// Mitsubishi GX Works2 project: ST_FB_NEW   PLC: Q02U

PROGRAM DIO
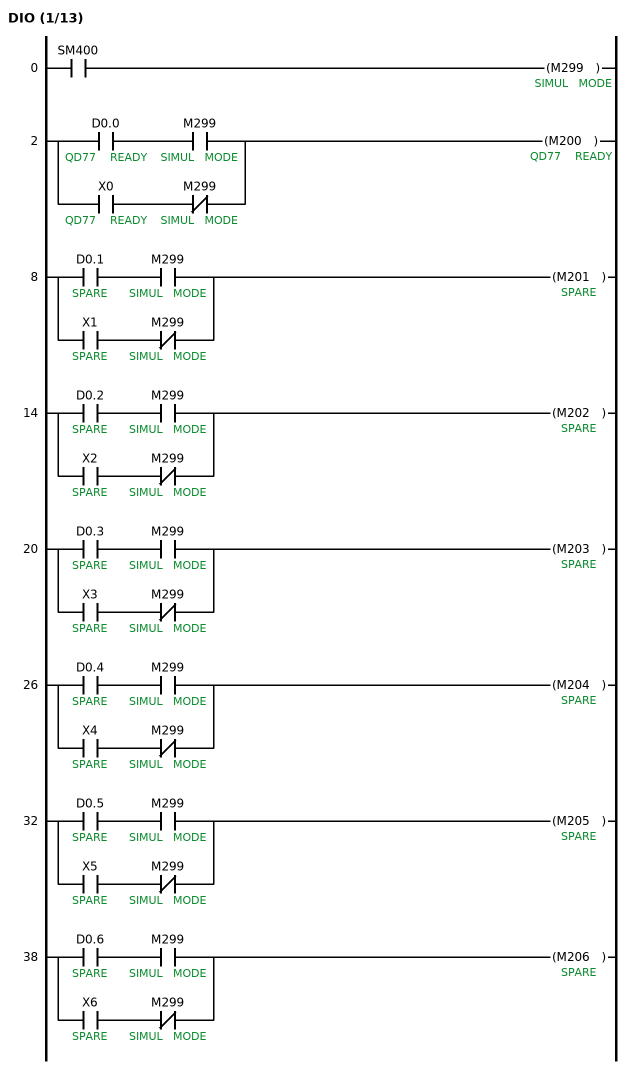
0     LD      SM400
      OUT     M299  ; SIMUL   MODE
2     LD      D0.0  ; QD77    READY
      AND     M299  ; SIMUL   MODE
      LD      X0  ; QD77    READY
      ANI     M299  ; SIMUL   MODE
      ORB
      OUT     M200  ; QD77    READY
8     LD      D0.1  ; SPARE
      AND     M299  ; SIMUL   MODE
      LD      X1  ; SPARE
      ANI     M299  ; SIMUL   MODE
      ORB
      OUT     M201  ; SPARE
14    LD      D0.2  ; SPARE
      AND     M299  ; SIMUL   MODE
      LD      X2  ; SPARE
      ANI     M299  ; SIMUL   MODE
      ORB
      OUT     M202  ; SPARE
20    LD      D0.3  ; SPARE
      AND     M299  ; SIMUL   MODE
      LD      X3  ; SPARE
      ANI     M299  ; SIMUL   MODE
      ORB
      OUT     M203  ; SPARE
26    LD      D0.4  ; SPARE
      AND     M299  ; SIMUL   MODE
      LD      X4  ; SPARE
      ANI     M299  ; SIMUL   MODE
      ORB
      OUT     M204  ; SPARE
32    LD      D0.5  ; SPARE
      AND     M299  ; SIMUL   MODE
      LD      X5  ; SPARE
      ANI     M299  ; SIMUL   MODE
      ORB
      OUT     M205  ; SPARE
38    LD      D0.6  ; SPARE
      AND     M299  ; SIMUL   MODE
      LD      X6  ; SPARE
      ANI     M299  ; SIMUL   MODE
      ORB
      OUT     M206  ; SPARE
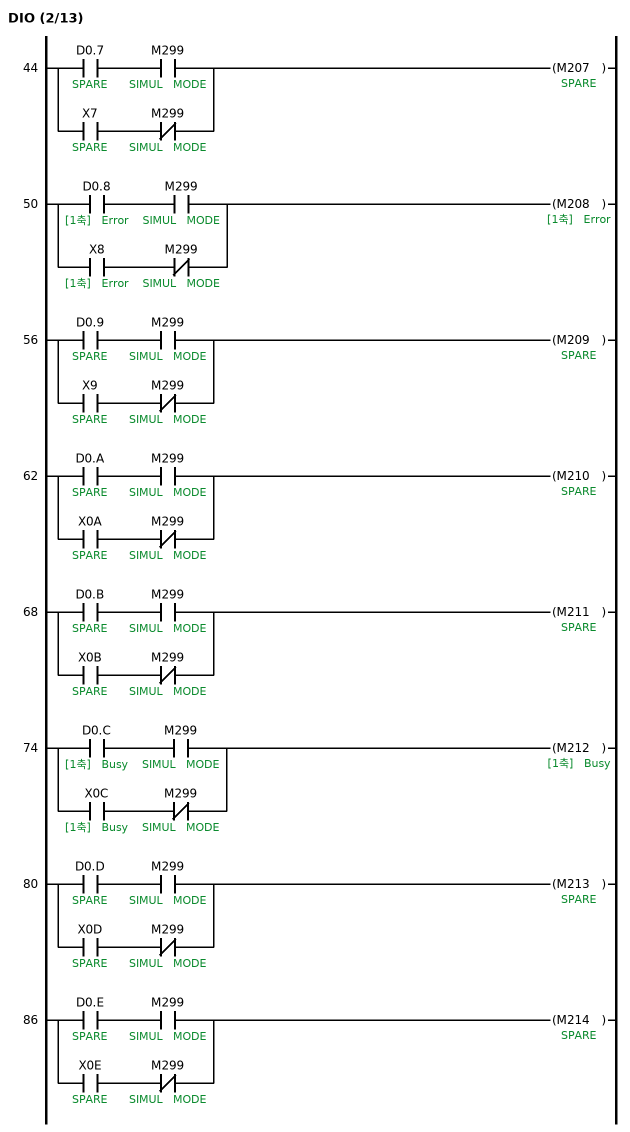
44    LD      D0.7  ; SPARE
      AND     M299  ; SIMUL   MODE
      LD      X7  ; SPARE
      ANI     M299  ; SIMUL   MODE
      ORB
      OUT     M207  ; SPARE
50    LD      D0.8  ; [1축]   Error
      AND     M299  ; SIMUL   MODE
      LD      X8  ; [1축]   Error
      ANI     M299  ; SIMUL   MODE
      ORB
      OUT     M208  ; [1축]   Error
56    LD      D0.9  ; SPARE
      AND     M299  ; SIMUL   MODE
      LD      X9  ; SPARE
      ANI     M299  ; SIMUL   MODE
      ORB
      OUT     M209  ; SPARE
62    LD      D0.A  ; SPARE
      AND     M299  ; SIMUL   MODE
      LD      X0A  ; SPARE
      ANI     M299  ; SIMUL   MODE
      ORB
      OUT     M210  ; SPARE
68    LD      D0.B  ; SPARE
      AND     M299  ; SIMUL   MODE
      LD      X0B  ; SPARE
      ANI     M299  ; SIMUL   MODE
      ORB
      OUT     M211  ; SPARE
74    LD      D0.C  ; [1축]   Busy
      AND     M299  ; SIMUL   MODE
      LD      X0C  ; [1축]   Busy
      ANI     M299  ; SIMUL   MODE
      ORB
      OUT     M212  ; [1축]   Busy
80    LD      D0.D  ; SPARE
      AND     M299  ; SIMUL   MODE
      LD      X0D  ; SPARE
      ANI     M299  ; SIMUL   MODE
      ORB
      OUT     M213  ; SPARE
86    LD      D0.E  ; SPARE
      AND     M299  ; SIMUL   MODE
      LD      X0E  ; SPARE
      ANI     M299  ; SIMUL   MODE
      ORB
      OUT     M214  ; SPARE
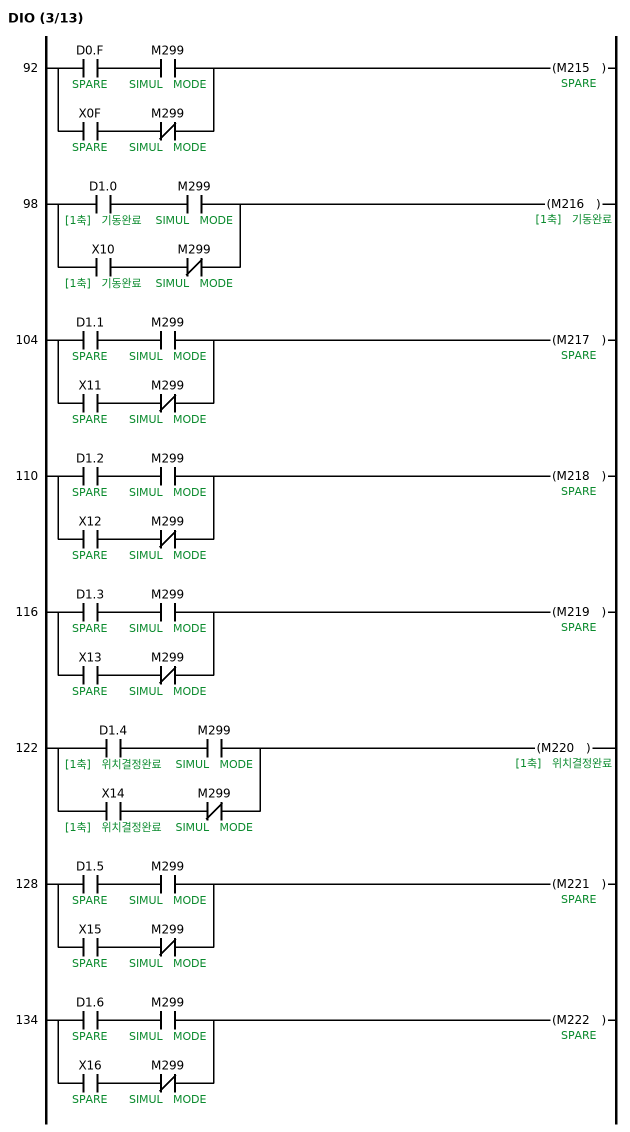
92    LD      D0.F  ; SPARE
      AND     M299  ; SIMUL   MODE
      LD      X0F  ; SPARE
      ANI     M299  ; SIMUL   MODE
      ORB
      OUT     M215  ; SPARE
98    LD      D1.0  ; [1축]   기동완료
      AND     M299  ; SIMUL   MODE
      LD      X10  ; [1축]   기동완료
      ANI     M299  ; SIMUL   MODE
      ORB
      OUT     M216  ; [1축]   기동완료
104   LD      D1.1  ; SPARE
      AND     M299  ; SIMUL   MODE
      LD      X11  ; SPARE
      ANI     M299  ; SIMUL   MODE
      ORB
      OUT     M217  ; SPARE
110   LD      D1.2  ; SPARE
      AND     M299  ; SIMUL   MODE
      LD      X12  ; SPARE
      ANI     M299  ; SIMUL   MODE
      ORB
      OUT     M218  ; SPARE
116   LD      D1.3  ; SPARE
      AND     M299  ; SIMUL   MODE
      LD      X13  ; SPARE
      ANI     M299  ; SIMUL   MODE
      ORB
      OUT     M219  ; SPARE
122   LD      D1.4  ; [1축]   위치결정완료
      AND     M299  ; SIMUL   MODE
      LD      X14  ; [1축]   위치결정완료
      ANI     M299  ; SIMUL   MODE
      ORB
      OUT     M220  ; [1축]   위치결정완료
128   LD      D1.5  ; SPARE
      AND     M299  ; SIMUL   MODE
      LD      X15  ; SPARE
      ANI     M299  ; SIMUL   MODE
      ORB
      OUT     M221  ; SPARE
134   LD      D1.6  ; SPARE
      AND     M299  ; SIMUL   MODE
      LD      X16  ; SPARE
      ANI     M299  ; SIMUL   MODE
      ORB
      OUT     M222  ; SPARE
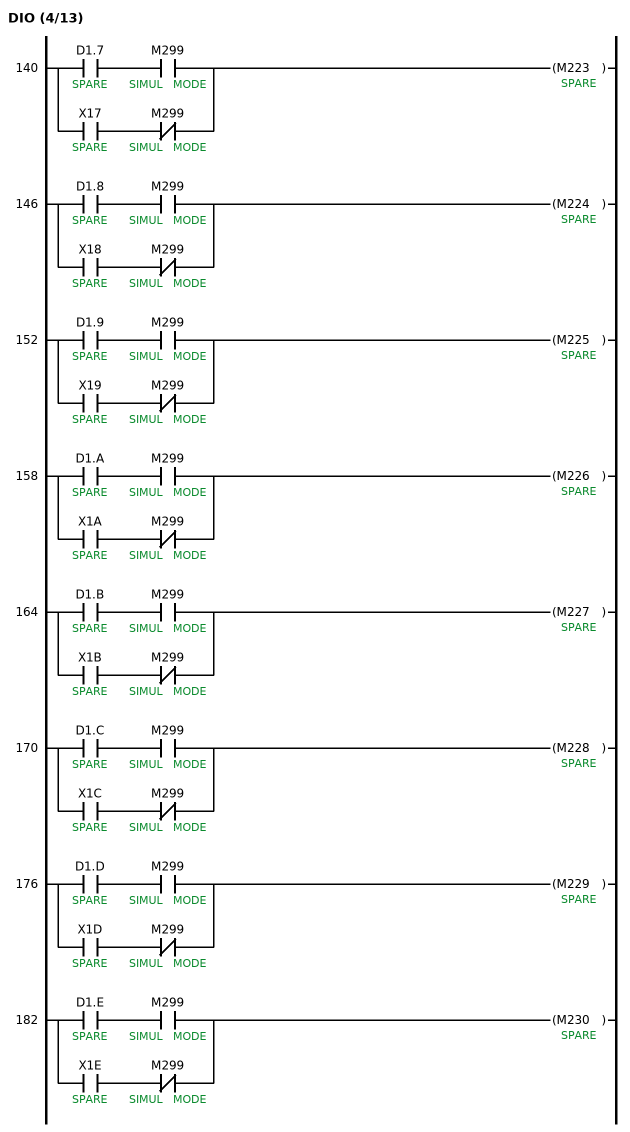
140   LD      D1.7  ; SPARE
      AND     M299  ; SIMUL   MODE
      LD      X17  ; SPARE
      ANI     M299  ; SIMUL   MODE
      ORB
      OUT     M223  ; SPARE
146   LD      D1.8  ; SPARE
      AND     M299  ; SIMUL   MODE
      LD      X18  ; SPARE
      ANI     M299  ; SIMUL   MODE
      ORB
      OUT     M224  ; SPARE
152   LD      D1.9  ; SPARE
      AND     M299  ; SIMUL   MODE
      LD      X19  ; SPARE
      ANI     M299  ; SIMUL   MODE
      ORB
      OUT     M225  ; SPARE
158   LD      D1.A  ; SPARE
      AND     M299  ; SIMUL   MODE
      LD      X1A  ; SPARE
      ANI     M299  ; SIMUL   MODE
      ORB
      OUT     M226  ; SPARE
164   LD      D1.B  ; SPARE
      AND     M299  ; SIMUL   MODE
      LD      X1B  ; SPARE
      ANI     M299  ; SIMUL   MODE
      ORB
      OUT     M227  ; SPARE
170   LD      D1.C  ; SPARE
      AND     M299  ; SIMUL   MODE
      LD      X1C  ; SPARE
      ANI     M299  ; SIMUL   MODE
      ORB
      OUT     M228  ; SPARE
176   LD      D1.D  ; SPARE
      AND     M299  ; SIMUL   MODE
      LD      X1D  ; SPARE
      ANI     M299  ; SIMUL   MODE
      ORB
      OUT     M229  ; SPARE
182   LD      D1.E  ; SPARE
      AND     M299  ; SIMUL   MODE
      LD      X1E  ; SPARE
      ANI     M299  ; SIMUL   MODE
      ORB
      OUT     M230  ; SPARE
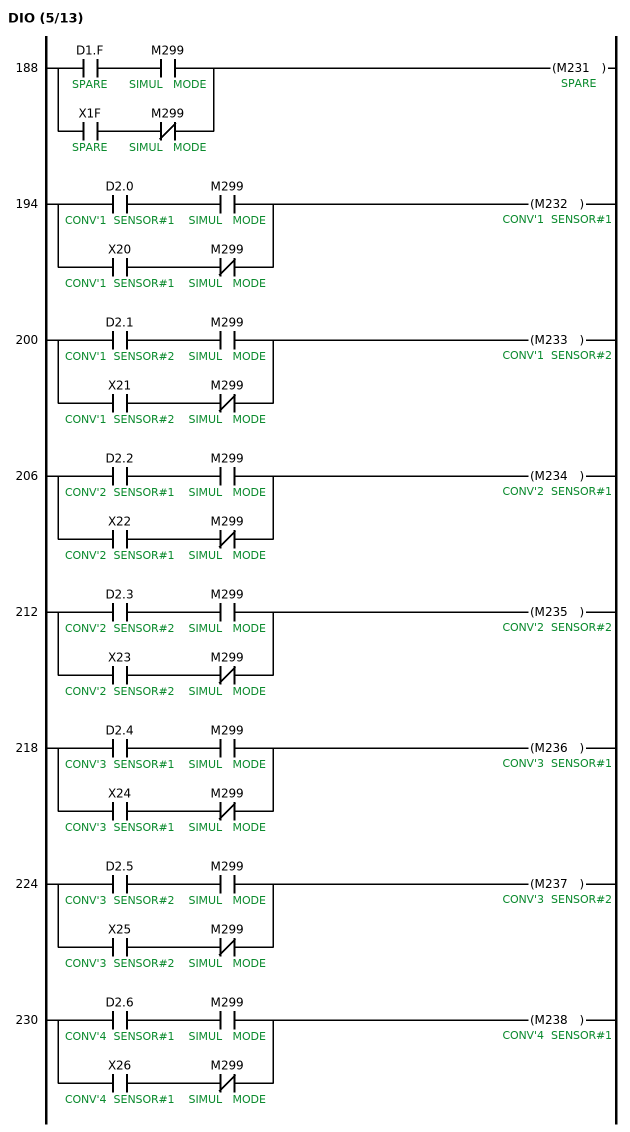
188   LD      D1.F  ; SPARE
      AND     M299  ; SIMUL   MODE
      LD      X1F  ; SPARE
      ANI     M299  ; SIMUL   MODE
      ORB
      OUT     M231  ; SPARE
194   LD      D2.0  ; CONV'1  SENSOR#1
      AND     M299  ; SIMUL   MODE
      LD      X20  ; CONV'1  SENSOR#1
      ANI     M299  ; SIMUL   MODE
      ORB
      OUT     M232  ; CONV'1  SENSOR#1
200   LD      D2.1  ; CONV'1  SENSOR#2
      AND     M299  ; SIMUL   MODE
      LD      X21  ; CONV'1  SENSOR#2
      ANI     M299  ; SIMUL   MODE
      ORB
      OUT     M233  ; CONV'1  SENSOR#2
206   LD      D2.2  ; CONV'2  SENSOR#1
      AND     M299  ; SIMUL   MODE
      LD      X22  ; CONV'2  SENSOR#1
      ANI     M299  ; SIMUL   MODE
      ORB
      OUT     M234  ; CONV'2  SENSOR#1
212   LD      D2.3  ; CONV'2  SENSOR#2
      AND     M299  ; SIMUL   MODE
      LD      X23  ; CONV'2  SENSOR#2
      ANI     M299  ; SIMUL   MODE
      ORB
      OUT     M235  ; CONV'2  SENSOR#2
218   LD      D2.4  ; CONV'3  SENSOR#1
      AND     M299  ; SIMUL   MODE
      LD      X24  ; CONV'3  SENSOR#1
      ANI     M299  ; SIMUL   MODE
      ORB
      OUT     M236  ; CONV'3  SENSOR#1
224   LD      D2.5  ; CONV'3  SENSOR#2
      AND     M299  ; SIMUL   MODE
      LD      X25  ; CONV'3  SENSOR#2
      ANI     M299  ; SIMUL   MODE
      ORB
      OUT     M237  ; CONV'3  SENSOR#2
230   LD      D2.6  ; CONV'4  SENSOR#1
      AND     M299  ; SIMUL   MODE
      LD      X26  ; CONV'4  SENSOR#1
      ANI     M299  ; SIMUL   MODE
      ORB
      OUT     M238  ; CONV'4  SENSOR#1
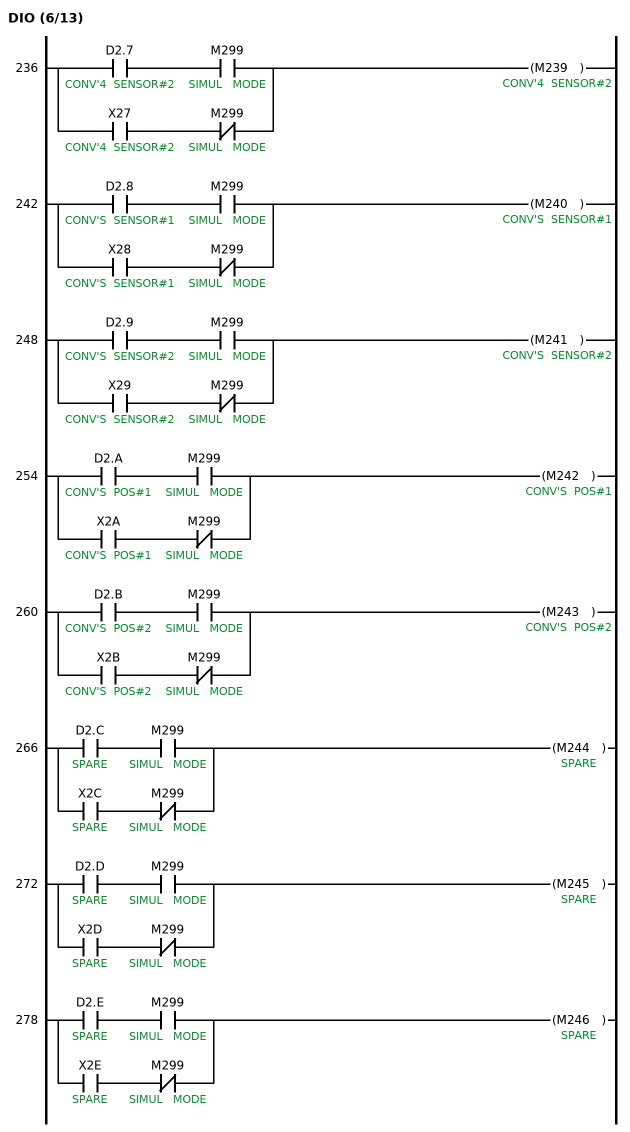
236   LD      D2.7  ; CONV'4  SENSOR#2
      AND     M299  ; SIMUL   MODE
      LD      X27  ; CONV'4  SENSOR#2
      ANI     M299  ; SIMUL   MODE
      ORB
      OUT     M239  ; CONV'4  SENSOR#2
242   LD      D2.8  ; CONV'S  SENSOR#1
      AND     M299  ; SIMUL   MODE
      LD      X28  ; CONV'S  SENSOR#1
      ANI     M299  ; SIMUL   MODE
      ORB
      OUT     M240  ; CONV'S  SENSOR#1
248   LD      D2.9  ; CONV'S  SENSOR#2
      AND     M299  ; SIMUL   MODE
      LD      X29  ; CONV'S  SENSOR#2
      ANI     M299  ; SIMUL   MODE
      ORB
      OUT     M241  ; CONV'S  SENSOR#2
254   LD      D2.A  ; CONV'S  POS#1
      AND     M299  ; SIMUL   MODE
      LD      X2A  ; CONV'S  POS#1
      ANI     M299  ; SIMUL   MODE
      ORB
      OUT     M242  ; CONV'S  POS#1
260   LD      D2.B  ; CONV'S  POS#2
      AND     M299  ; SIMUL   MODE
      LD      X2B  ; CONV'S  POS#2
      ANI     M299  ; SIMUL   MODE
      ORB
      OUT     M243  ; CONV'S  POS#2
266   LD      D2.C  ; SPARE
      AND     M299  ; SIMUL   MODE
      LD      X2C  ; SPARE
      ANI     M299  ; SIMUL   MODE
      ORB
      OUT     M244  ; SPARE
272   LD      D2.D  ; SPARE
      AND     M299  ; SIMUL   MODE
      LD      X2D  ; SPARE
      ANI     M299  ; SIMUL   MODE
      ORB
      OUT     M245  ; SPARE
278   LD      D2.E  ; SPARE
      AND     M299  ; SIMUL   MODE
      LD      X2E  ; SPARE
      ANI     M299  ; SIMUL   MODE
      ORB
      OUT     M246  ; SPARE
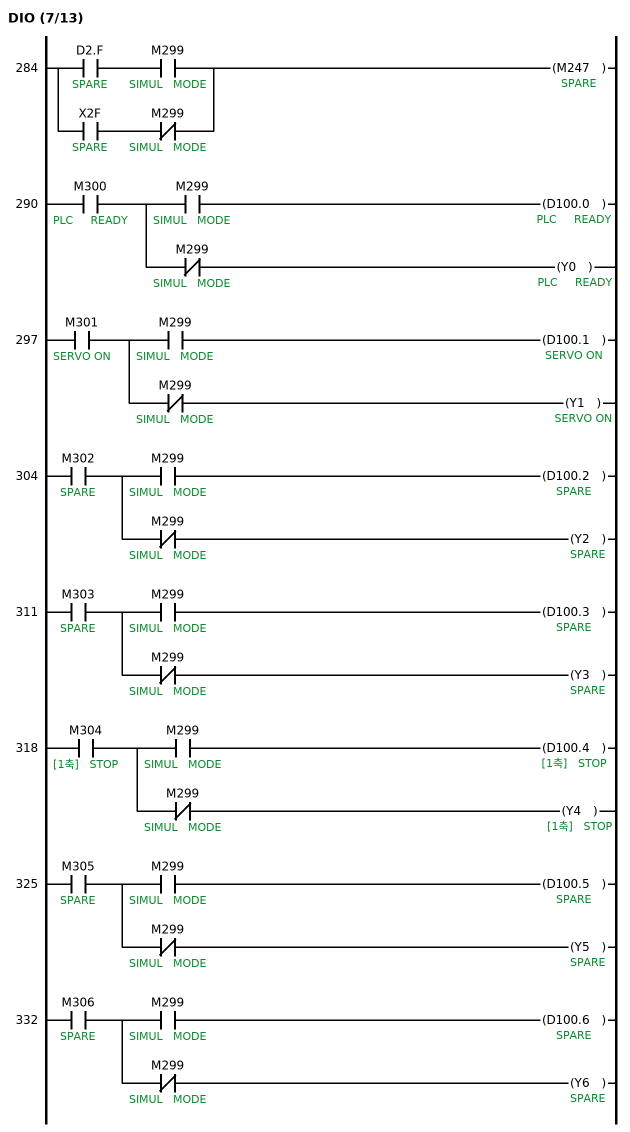
284   LD      D2.F  ; SPARE
      AND     M299  ; SIMUL   MODE
      LD      X2F  ; SPARE
      ANI     M299  ; SIMUL   MODE
      ORB
      OUT     M247  ; SPARE
290   LD      M300  ; PLC     READY
      MPS
      AND     M299  ; SIMUL   MODE
      OUT     D100.0  ; PLC     READY
      MPP
      ANI     M299  ; SIMUL   MODE
      OUT     Y0  ; PLC     READY
297   LD      M301  ; SERVO ON
      MPS
      AND     M299  ; SIMUL   MODE
      OUT     D100.1  ; SERVO ON
      MPP
      ANI     M299  ; SIMUL   MODE
      OUT     Y1  ; SERVO ON
304   LD      M302  ; SPARE
      MPS
      AND     M299  ; SIMUL   MODE
      OUT     D100.2  ; SPARE
      MPP
      ANI     M299  ; SIMUL   MODE
      OUT     Y2  ; SPARE
311   LD      M303  ; SPARE
      MPS
      AND     M299  ; SIMUL   MODE
      OUT     D100.3  ; SPARE
      MPP
      ANI     M299  ; SIMUL   MODE
      OUT     Y3  ; SPARE
318   LD      M304  ; [1축]   STOP
      MPS
      AND     M299  ; SIMUL   MODE
      OUT     D100.4  ; [1축]   STOP
      MPP
      ANI     M299  ; SIMUL   MODE
      OUT     Y4  ; [1축]   STOP
325   LD      M305  ; SPARE
      MPS
      AND     M299  ; SIMUL   MODE
      OUT     D100.5  ; SPARE
      MPP
      ANI     M299  ; SIMUL   MODE
      OUT     Y5  ; SPARE
332   LD      M306  ; SPARE
      MPS
      AND     M299  ; SIMUL   MODE
      OUT     D100.6  ; SPARE
      MPP
      ANI     M299  ; SIMUL   MODE
      OUT     Y6  ; SPARE
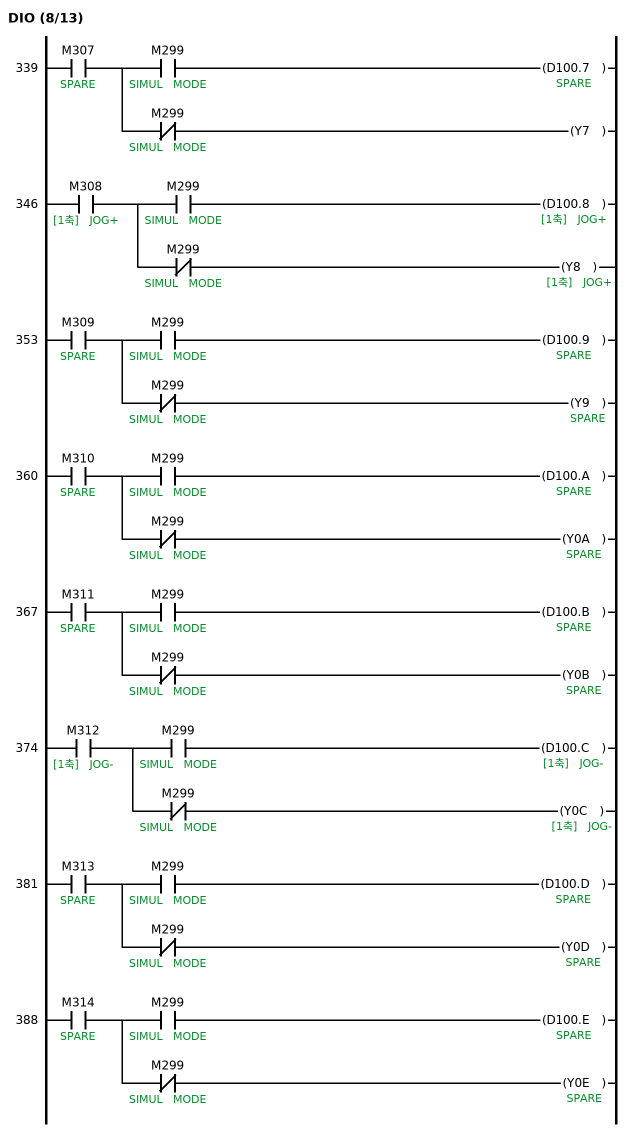
339   LD      M307  ; SPARE
      MPS
      AND     M299  ; SIMUL   MODE
      OUT     D100.7  ; SPARE
      MPP
      ANI     M299  ; SIMUL   MODE
      OUT     Y7
346   LD      M308  ; [1축]   JOG+
      MPS
      AND     M299  ; SIMUL   MODE
      OUT     D100.8  ; [1축]   JOG+
      MPP
      ANI     M299  ; SIMUL   MODE
      OUT     Y8  ; [1축]   JOG+
353   LD      M309  ; SPARE
      MPS
      AND     M299  ; SIMUL   MODE
      OUT     D100.9  ; SPARE
      MPP
      ANI     M299  ; SIMUL   MODE
      OUT     Y9  ; SPARE
360   LD      M310  ; SPARE
      MPS
      AND     M299  ; SIMUL   MODE
      OUT     D100.A  ; SPARE
      MPP
      ANI     M299  ; SIMUL   MODE
      OUT     Y0A  ; SPARE
367   LD      M311  ; SPARE
      MPS
      AND     M299  ; SIMUL   MODE
      OUT     D100.B  ; SPARE
      MPP
      ANI     M299  ; SIMUL   MODE
      OUT     Y0B  ; SPARE
374   LD      M312  ; [1축]   JOG-
      MPS
      AND     M299  ; SIMUL   MODE
      OUT     D100.C  ; [1축]   JOG-
      MPP
      ANI     M299  ; SIMUL   MODE
      OUT     Y0C  ; [1축]   JOG-
381   LD      M313  ; SPARE
      MPS
      AND     M299  ; SIMUL   MODE
      OUT     D100.D  ; SPARE
      MPP
      ANI     M299  ; SIMUL   MODE
      OUT     Y0D  ; SPARE
388   LD      M314  ; SPARE
      MPS
      AND     M299  ; SIMUL   MODE
      OUT     D100.E  ; SPARE
      MPP
      ANI     M299  ; SIMUL   MODE
      OUT     Y0E  ; SPARE
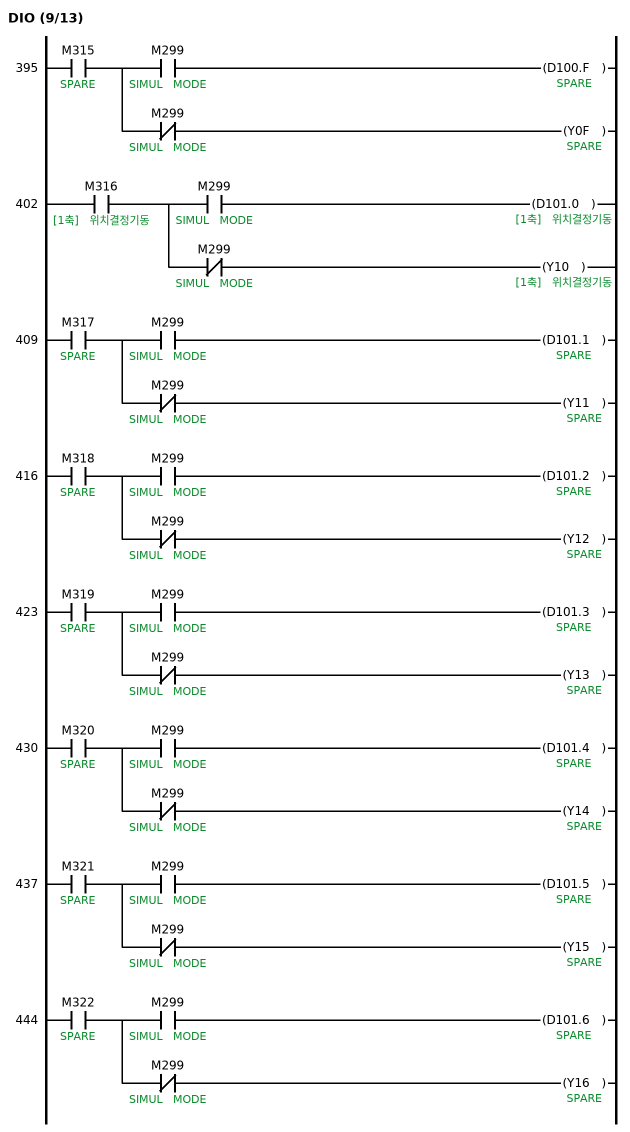
395   LD      M315  ; SPARE
      MPS
      AND     M299  ; SIMUL   MODE
      OUT     D100.F  ; SPARE
      MPP
      ANI     M299  ; SIMUL   MODE
      OUT     Y0F  ; SPARE
402   LD      M316  ; [1축]   위치결정기동
      MPS
      AND     M299  ; SIMUL   MODE
      OUT     D101.0  ; [1축]   위치결정기동
      MPP
      ANI     M299  ; SIMUL   MODE
      OUT     Y10  ; [1축]   위치결정기동
409   LD      M317  ; SPARE
      MPS
      AND     M299  ; SIMUL   MODE
      OUT     D101.1  ; SPARE
      MPP
      ANI     M299  ; SIMUL   MODE
      OUT     Y11  ; SPARE
416   LD      M318  ; SPARE
      MPS
      AND     M299  ; SIMUL   MODE
      OUT     D101.2  ; SPARE
      MPP
      ANI     M299  ; SIMUL   MODE
      OUT     Y12  ; SPARE
423   LD      M319  ; SPARE
      MPS
      AND     M299  ; SIMUL   MODE
      OUT     D101.3  ; SPARE
      MPP
      ANI     M299  ; SIMUL   MODE
      OUT     Y13  ; SPARE
430   LD      M320  ; SPARE
      MPS
      AND     M299  ; SIMUL   MODE
      OUT     D101.4  ; SPARE
      MPP
      ANI     M299  ; SIMUL   MODE
      OUT     Y14  ; SPARE
437   LD      M321  ; SPARE
      MPS
      AND     M299  ; SIMUL   MODE
      OUT     D101.5  ; SPARE
      MPP
      ANI     M299  ; SIMUL   MODE
      OUT     Y15  ; SPARE
444   LD      M322  ; SPARE
      MPS
      AND     M299  ; SIMUL   MODE
      OUT     D101.6  ; SPARE
      MPP
      ANI     M299  ; SIMUL   MODE
      OUT     Y16  ; SPARE
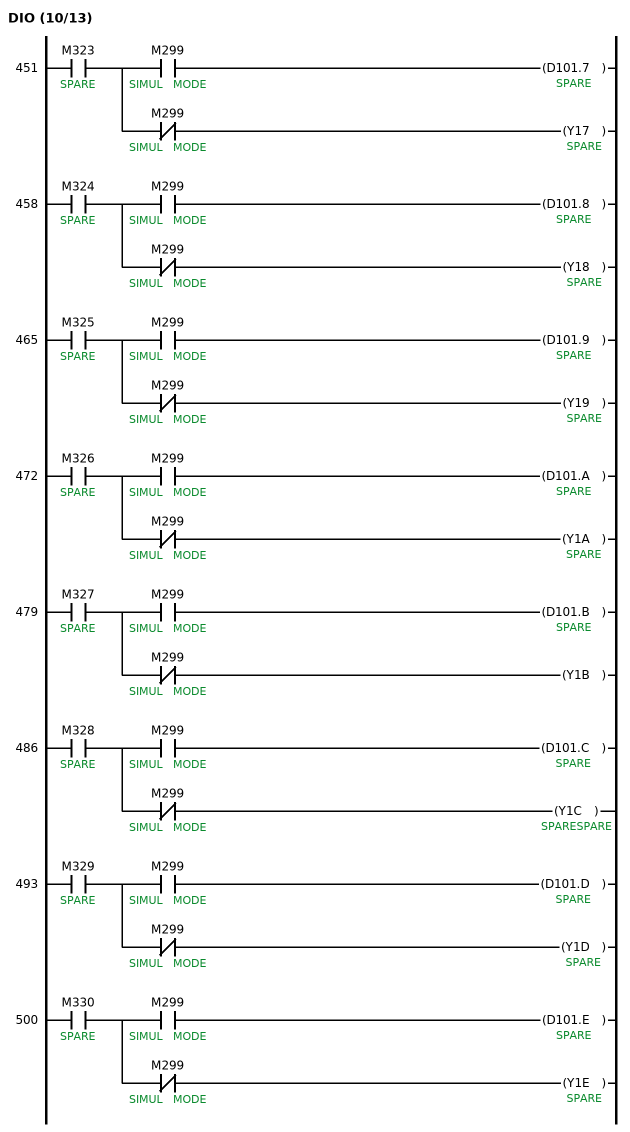
451   LD      M323  ; SPARE
      MPS
      AND     M299  ; SIMUL   MODE
      OUT     D101.7  ; SPARE
      MPP
      ANI     M299  ; SIMUL   MODE
      OUT     Y17  ; SPARE
458   LD      M324  ; SPARE
      MPS
      AND     M299  ; SIMUL   MODE
      OUT     D101.8  ; SPARE
      MPP
      ANI     M299  ; SIMUL   MODE
      OUT     Y18  ; SPARE
465   LD      M325  ; SPARE
      MPS
      AND     M299  ; SIMUL   MODE
      OUT     D101.9  ; SPARE
      MPP
      ANI     M299  ; SIMUL   MODE
      OUT     Y19  ; SPARE
472   LD      M326  ; SPARE
      MPS
      AND     M299  ; SIMUL   MODE
      OUT     D101.A  ; SPARE
      MPP
      ANI     M299  ; SIMUL   MODE
      OUT     Y1A  ; SPARE
479   LD      M327  ; SPARE
      MPS
      AND     M299  ; SIMUL   MODE
      OUT     D101.B  ; SPARE
      MPP
      ANI     M299  ; SIMUL   MODE
      OUT     Y1B
486   LD      M328  ; SPARE
      MPS
      AND     M299  ; SIMUL   MODE
      OUT     D101.C  ; SPARE
      MPP
      ANI     M299  ; SIMUL   MODE
      OUT     Y1C  ; SPARESPARE
493   LD      M329  ; SPARE
      MPS
      AND     M299  ; SIMUL   MODE
      OUT     D101.D  ; SPARE
      MPP
      ANI     M299  ; SIMUL   MODE
      OUT     Y1D  ; SPARE
500   LD      M330  ; SPARE
      MPS
      AND     M299  ; SIMUL   MODE
      OUT     D101.E  ; SPARE
      MPP
      ANI     M299  ; SIMUL   MODE
      OUT     Y1E  ; SPARE
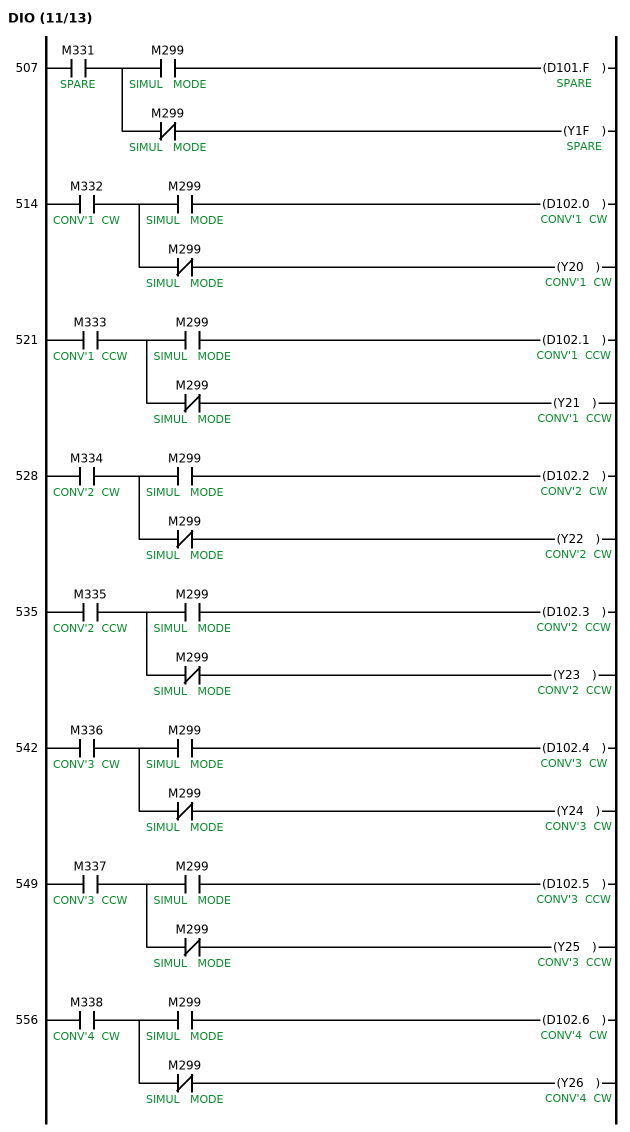
507   LD      M331  ; SPARE
      MPS
      AND     M299  ; SIMUL   MODE
      OUT     D101.F  ; SPARE
      MPP
      ANI     M299  ; SIMUL   MODE
      OUT     Y1F  ; SPARE
514   LD      M332  ; CONV'1  CW
      MPS
      AND     M299  ; SIMUL   MODE
      OUT     D102.0  ; CONV'1  CW
      MPP
      ANI     M299  ; SIMUL   MODE
      OUT     Y20  ; CONV'1  CW
521   LD      M333  ; CONV'1  CCW
      MPS
      AND     M299  ; SIMUL   MODE
      OUT     D102.1  ; CONV'1  CCW
      MPP
      ANI     M299  ; SIMUL   MODE
      OUT     Y21  ; CONV'1  CCW
528   LD      M334  ; CONV'2  CW
      MPS
      AND     M299  ; SIMUL   MODE
      OUT     D102.2  ; CONV'2  CW
      MPP
      ANI     M299  ; SIMUL   MODE
      OUT     Y22  ; CONV'2  CW
535   LD      M335  ; CONV'2  CCW
      MPS
      AND     M299  ; SIMUL   MODE
      OUT     D102.3  ; CONV'2  CCW
      MPP
      ANI     M299  ; SIMUL   MODE
      OUT     Y23  ; CONV'2  CCW
542   LD      M336  ; CONV'3  CW
      MPS
      AND     M299  ; SIMUL   MODE
      OUT     D102.4  ; CONV'3  CW
      MPP
      ANI     M299  ; SIMUL   MODE
      OUT     Y24  ; CONV'3  CW
549   LD      M337  ; CONV'3  CCW
      MPS
      AND     M299  ; SIMUL   MODE
      OUT     D102.5  ; CONV'3  CCW
      MPP
      ANI     M299  ; SIMUL   MODE
      OUT     Y25  ; CONV'3  CCW
556   LD      M338  ; CONV'4  CW
      MPS
      AND     M299  ; SIMUL   MODE
      OUT     D102.6  ; CONV'4  CW
      MPP
      ANI     M299  ; SIMUL   MODE
      OUT     Y26  ; CONV'4  CW
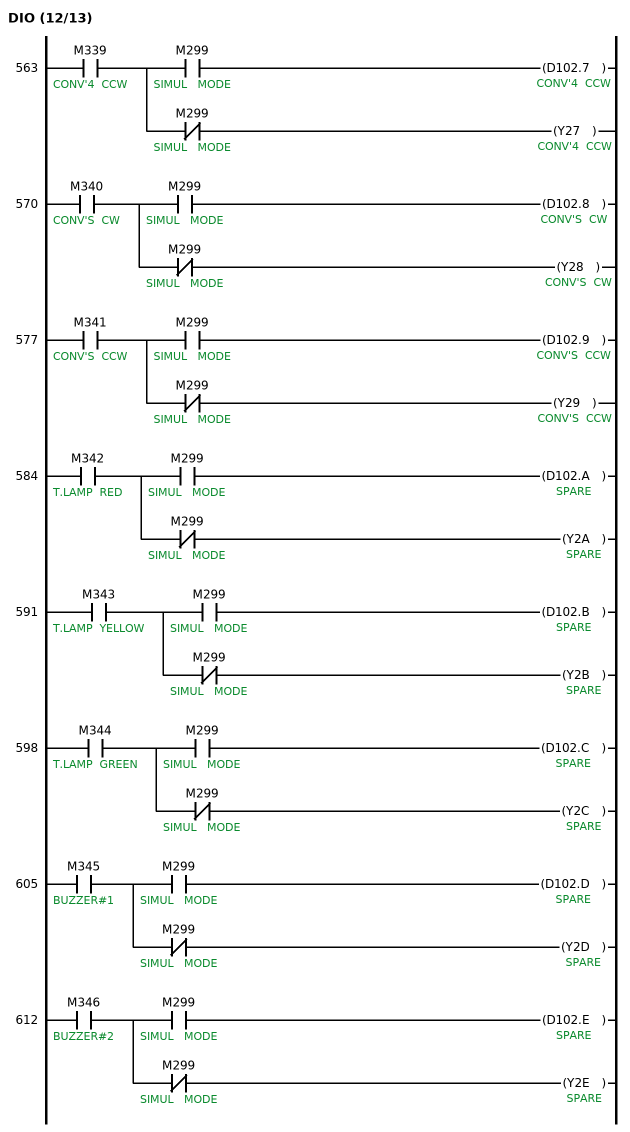
563   LD      M339  ; CONV'4  CCW
      MPS
      AND     M299  ; SIMUL   MODE
      OUT     D102.7  ; CONV'4  CCW
      MPP
      ANI     M299  ; SIMUL   MODE
      OUT     Y27  ; CONV'4  CCW
570   LD      M340  ; CONV'S  CW
      MPS
      AND     M299  ; SIMUL   MODE
      OUT     D102.8  ; CONV'S  CW
      MPP
      ANI     M299  ; SIMUL   MODE
      OUT     Y28  ; CONV'S  CW
577   LD      M341  ; CONV'S  CCW
      MPS
      AND     M299  ; SIMUL   MODE
      OUT     D102.9  ; CONV'S  CCW
      MPP
      ANI     M299  ; SIMUL   MODE
      OUT     Y29  ; CONV'S  CCW
584   LD      M342  ; T.LAMP  RED
      MPS
      AND     M299  ; SIMUL   MODE
      OUT     D102.A  ; SPARE
      MPP
      ANI     M299  ; SIMUL   MODE
      OUT     Y2A  ; SPARE
591   LD      M343  ; T.LAMP  YELLOW
      MPS
      AND     M299  ; SIMUL   MODE
      OUT     D102.B  ; SPARE
      MPP
      ANI     M299  ; SIMUL   MODE
      OUT     Y2B  ; SPARE
598   LD      M344  ; T.LAMP  GREEN
      MPS
      AND     M299  ; SIMUL   MODE
      OUT     D102.C  ; SPARE
      MPP
      ANI     M299  ; SIMUL   MODE
      OUT     Y2C  ; SPARE
605   LD      M345  ; BUZZER#1
      MPS
      AND     M299  ; SIMUL   MODE
      OUT     D102.D  ; SPARE
      MPP
      ANI     M299  ; SIMUL   MODE
      OUT     Y2D  ; SPARE
612   LD      M346  ; BUZZER#2
      MPS
      AND     M299  ; SIMUL   MODE
      OUT     D102.E  ; SPARE
      MPP
      ANI     M299  ; SIMUL   MODE
      OUT     Y2E  ; SPARE
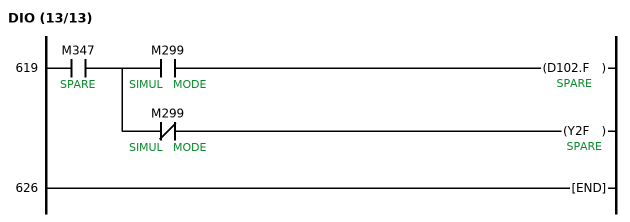
619   LD      M347  ; SPARE
      MPS
      AND     M299  ; SIMUL   MODE
      OUT     D102.F  ; SPARE
      MPP
      ANI     M299  ; SIMUL   MODE
      OUT     Y2F  ; SPARE
626   END
END_PROGRAM

PROGRAM SERVO
VAR
  SERVO_FB_1 : SERVO_FB;
END_VAR
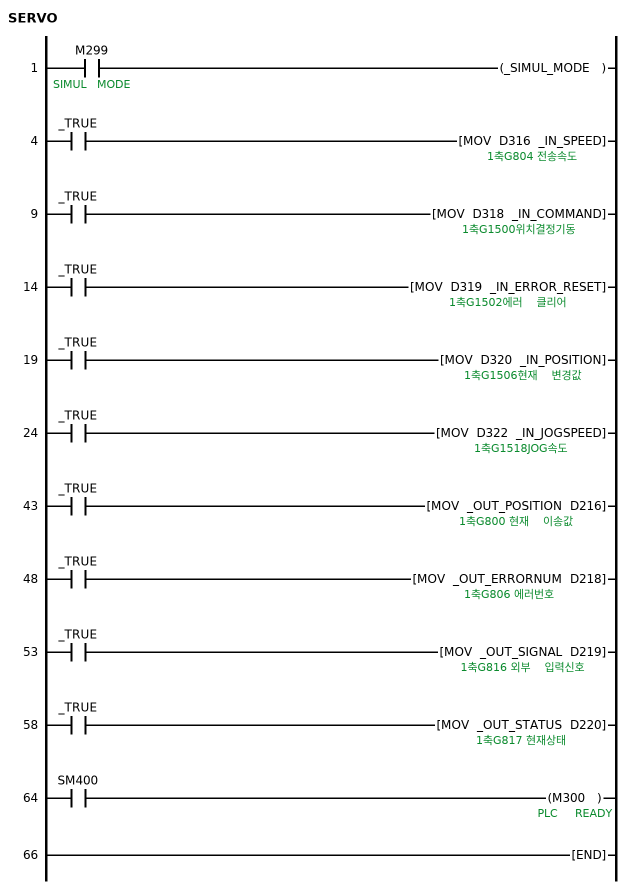
; FB BLK START SERVO_FB(SERVO_FB_1)
1     LD      M299  ; SIMUL   MODE
      OUT     _SIMUL_MODE
4     LD      _TRUE
      MOV     D316 _IN_SPEED  ; 1축G804 전송속도
9     LD      _TRUE
      MOV     D318 _IN_COMMAND  ; 1축G1500위치결정기동
14    LD      _TRUE
      MOV     D319 _IN_ERROR_RESET  ; 1축G1502에러    클리어
19    LD      _TRUE
      MOV     D320 _IN_POSITION  ; 1축G1506현재    변경값
24    LD      _TRUE
      MOV     D322 _IN_JOGSPEED  ; 1축G1518JOG속도
; FB START
; FB_NAME SERVO_FB
; INSTANCE_NAME SERVO_FB_1
; FB IN_B:SIMUL_MODE
; FB OUT_OUT_POSITION:W
; FB IN_W:IN_SPEED
; FB OUT_OUT_ERRORNUM:W
; FB IN_W:IN_COMMAND
; FB OUT_OUT_SIGNAL:W
; FB IN_W:IN_ERROR_RESET
; FB OUT_OUT_STATUS:W
; FB IN_W:IN_POSITION
; FB IN_W:IN_JOGSPEED
; FB END
43    LD      _TRUE
      MOV     _OUT_POSITION D216  ; 1축G800 현재    이송값
48    LD      _TRUE
      MOV     _OUT_ERRORNUM D218  ; 1축G806 에러번호
53    LD      _TRUE
      MOV     _OUT_SIGNAL D219  ; 1축G816 외부    입력신호
58    LD      _TRUE
      MOV     _OUT_STATUS D220  ; 1축G817 현재상태
; FB BLK END
64    LD      SM400
      OUT     M300  ; PLC     READY
66    END
END_PROGRAM

PROGRAM MODE
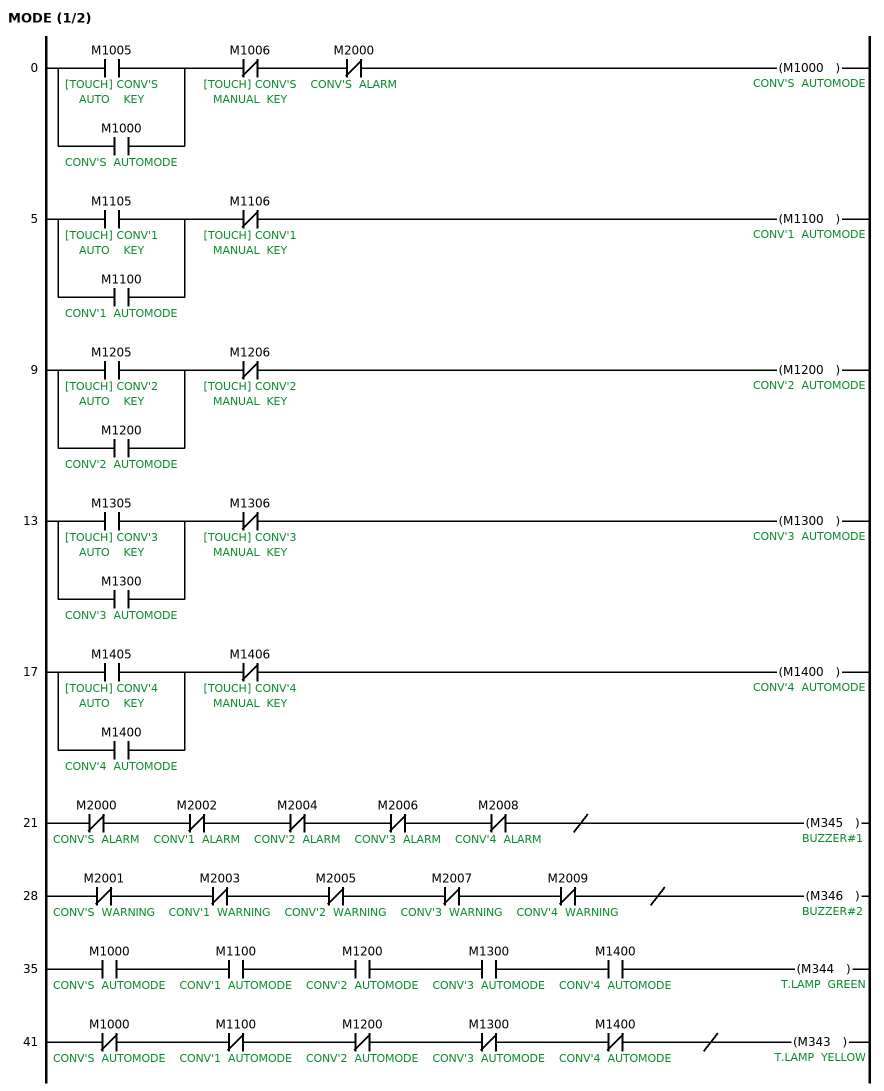
0     LD      M1005  ; [TOUCH] CONV'S  AUTO    KEY
      OR      M1000  ; CONV'S  AUTOMODE
      ANI     M1006  ; [TOUCH] CONV'S  MANUAL  KEY
      ANI     M2000  ; CONV'S  ALARM
      OUT     M1000  ; CONV'S  AUTOMODE
5     LD      M1105  ; [TOUCH] CONV'1  AUTO    KEY
      OR      M1100  ; CONV'1  AUTOMODE
      ANI     M1106  ; [TOUCH] CONV'1  MANUAL  KEY
      OUT     M1100  ; CONV'1  AUTOMODE
9     LD      M1205  ; [TOUCH] CONV'2  AUTO    KEY
      OR      M1200  ; CONV'2  AUTOMODE
      ANI     M1206  ; [TOUCH] CONV'2  MANUAL  KEY
      OUT     M1200  ; CONV'2  AUTOMODE
13    LD      M1305  ; [TOUCH] CONV'3  AUTO    KEY
      OR      M1300  ; CONV'3  AUTOMODE
      ANI     M1306  ; [TOUCH] CONV'3  MANUAL  KEY
      OUT     M1300  ; CONV'3  AUTOMODE
17    LD      M1405  ; [TOUCH] CONV'4  AUTO    KEY
      OR      M1400  ; CONV'4  AUTOMODE
      ANI     M1406  ; [TOUCH] CONV'4  MANUAL  KEY
      OUT     M1400  ; CONV'4  AUTOMODE
21    LDI     M2000  ; CONV'S  ALARM
      ANI     M2002  ; CONV'1  ALARM
      ANI     M2004  ; CONV'2  ALARM
      ANI     M2006  ; CONV'3  ALARM
      ANI     M2008  ; CONV'4  ALARM
      INV
      OUT     M345  ; BUZZER#1
28    LDI     M2001  ; CONV'S  WARNING
      ANI     M2003  ; CONV'1  WARNING
      ANI     M2005  ; CONV'2  WARNING
      ANI     M2007  ; CONV'3  WARNING
      ANI     M2009  ; CONV'4  WARNING
      INV
      OUT     M346  ; BUZZER#2
35    LD      M1000  ; CONV'S  AUTOMODE
      AND     M1100  ; CONV'1  AUTOMODE
      AND     M1200  ; CONV'2  AUTOMODE
      AND     M1300  ; CONV'3  AUTOMODE
      AND     M1400  ; CONV'4  AUTOMODE
      OUT     M344  ; T.LAMP  GREEN
41    LDI     M1000  ; CONV'S  AUTOMODE
      ANI     M1100  ; CONV'1  AUTOMODE
      ANI     M1200  ; CONV'2  AUTOMODE
      ANI     M1300  ; CONV'3  AUTOMODE
      ANI     M1400  ; CONV'4  AUTOMODE
      INV
      OUT     M343  ; T.LAMP  YELLOW
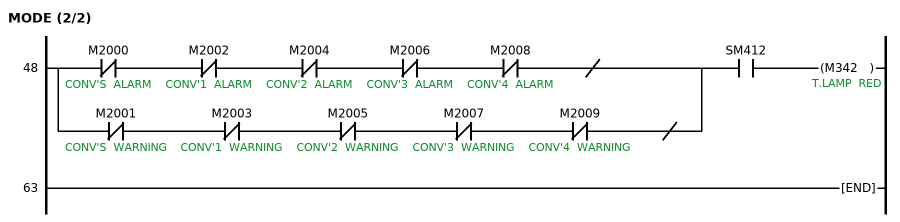
48    LDI     M2000  ; CONV'S  ALARM
      ANI     M2002  ; CONV'1  ALARM
      ANI     M2004  ; CONV'2  ALARM
      ANI     M2006  ; CONV'3  ALARM
      ANI     M2008  ; CONV'4  ALARM
      INV
      LDI     M2001  ; CONV'S  WARNING
      ANI     M2003  ; CONV'1  WARNING
      ANI     M2005  ; CONV'2  WARNING
      ANI     M2007  ; CONV'3  WARNING
      ANI     M2009  ; CONV'4  WARNING
      INV
      ORB
      AND     SM412
      OUT     M342  ; T.LAMP  RED
63    END
END_PROGRAM

PROGRAM CONVS
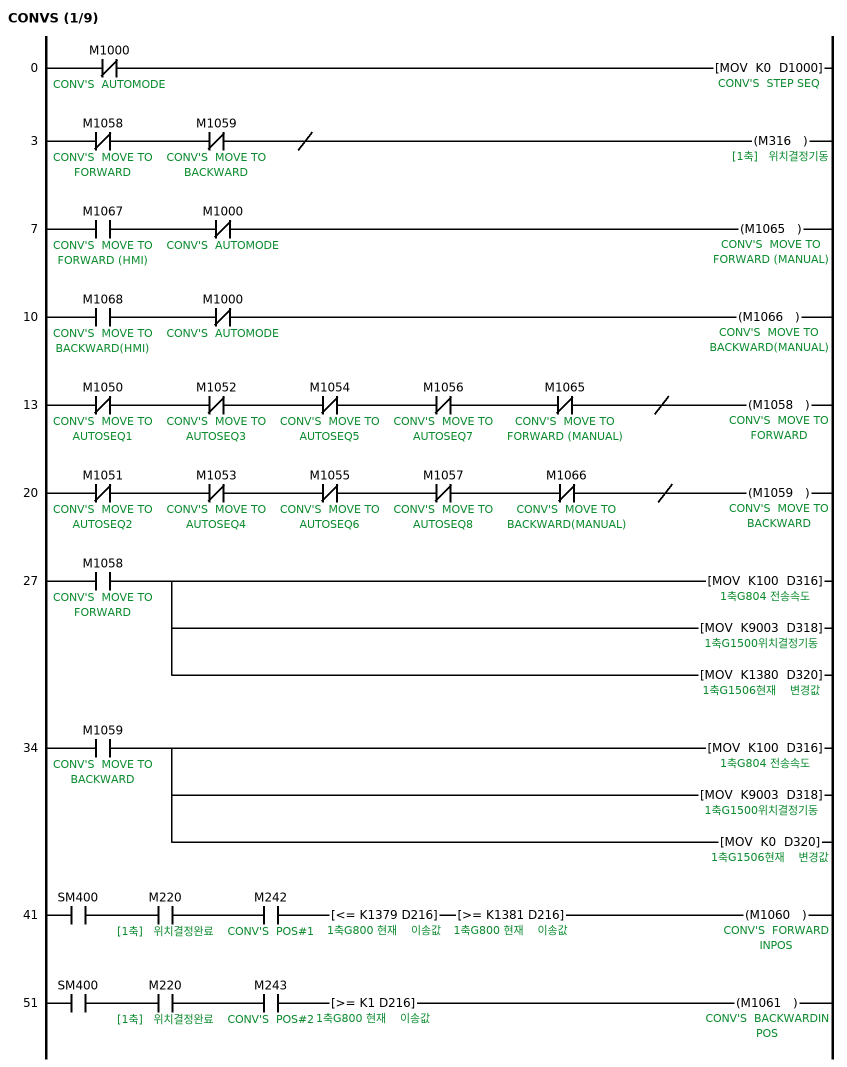
0     LDI     M1000  ; CONV'S  AUTOMODE
      MOV     K0 D1000  ; CONV'S  STEP SEQ
3     LDI     M1058  ; CONV'S  MOVE TO FORWARD
      ANI     M1059  ; CONV'S  MOVE TO BACKWARD
      INV
      OUT     M316  ; [1축]   위치결정기동
7     LD      M1067  ; CONV'S  MOVE TO FORWARD (HMI)
      ANI     M1000  ; CONV'S  AUTOMODE
      OUT     M1065  ; CONV'S  MOVE TO FORWARD (MANUAL)
10    LD      M1068  ; CONV'S  MOVE TO BACKWARD(HMI)
      ANI     M1000  ; CONV'S  AUTOMODE
      OUT     M1066  ; CONV'S  MOVE TO BACKWARD(MANUAL)
13    LDI     M1050  ; CONV'S  MOVE TO AUTOSEQ1
      ANI     M1052  ; CONV'S  MOVE TO AUTOSEQ3
      ANI     M1054  ; CONV'S  MOVE TO AUTOSEQ5
      ANI     M1056  ; CONV'S  MOVE TO AUTOSEQ7
      ANI     M1065  ; CONV'S  MOVE TO FORWARD (MANUAL)
      INV
      OUT     M1058  ; CONV'S  MOVE TO FORWARD
20    LDI     M1051  ; CONV'S  MOVE TO AUTOSEQ2
      ANI     M1053  ; CONV'S  MOVE TO AUTOSEQ4
      ANI     M1055  ; CONV'S  MOVE TO AUTOSEQ6
      ANI     M1057  ; CONV'S  MOVE TO AUTOSEQ8
      ANI     M1066  ; CONV'S  MOVE TO BACKWARD(MANUAL)
      INV
      OUT     M1059  ; CONV'S  MOVE TO BACKWARD
27    LD      M1058  ; CONV'S  MOVE TO FORWARD
      MOV     K100 D316  ; 1축G804 전송속도
      MOV     K9003 D318  ; 1축G1500위치결정기동
      MOV     K1380 D320  ; 1축G1506현재    변경값
34    LD      M1059  ; CONV'S  MOVE TO BACKWARD
      MOV     K100 D316
      MOV     K9003 D318
      MOV     K0 D320
41    LD      SM400
      AND     M220  ; [1축]   위치결정완료
      AND     M242  ; CONV'S  POS#1
      AND<=   K1379 D216  ; 1축G800 현재    이송값
      AND>=   K1381 D216  ; 1축G800 현재    이송값
      OUT     M1060  ; CONV'S  FORWARD INPOS
51    LD      SM400
      AND     M220  ; [1축]   위치결정완료
      AND     M243  ; CONV'S  POS#2
      AND>=   K1 D216  ; 1축G800 현재    이송값
      OUT     M1061  ; CONV'S  BACKWARDINPOS
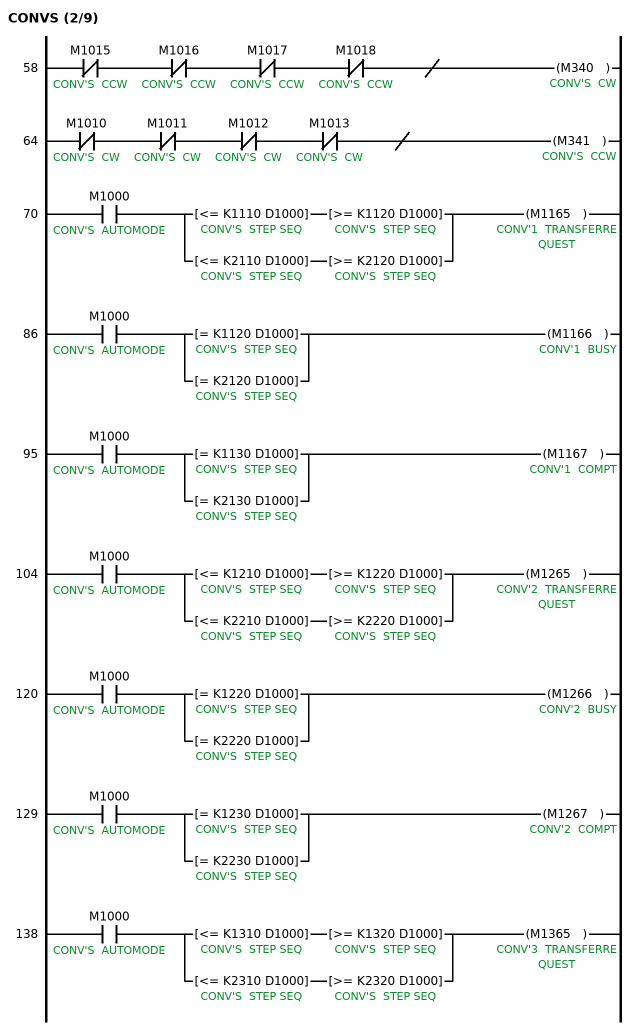
58    LDI     M1015  ; CONV'S  CCW
      ANI     M1016  ; CONV'S  CCW
      ANI     M1017  ; CONV'S  CCW
      ANI     M1018  ; CONV'S  CCW
      INV
      OUT     M340  ; CONV'S  CW
64    LDI     M1010  ; CONV'S  CW
      ANI     M1011  ; CONV'S  CW
      ANI     M1012  ; CONV'S  CW
      ANI     M1013  ; CONV'S  CW
      INV
      OUT     M341  ; CONV'S  CCW
70    LD      M1000  ; CONV'S  AUTOMODE
      LD<=    K1110 D1000  ; CONV'S  STEP SEQ
      AND>=   K1120 D1000  ; CONV'S  STEP SEQ
      LD<=    K2110 D1000  ; CONV'S  STEP SEQ
      AND>=   K2120 D1000  ; CONV'S  STEP SEQ
      ORB
      ANB
      OUT     M1165  ; CONV'1  TRANSFERREQUEST
86    LD      M1000  ; CONV'S  AUTOMODE
      LD=     K1120 D1000  ; CONV'S  STEP SEQ
      OR=     K2120 D1000  ; CONV'S  STEP SEQ
      ANB
      OUT     M1166  ; CONV'1  BUSY
95    LD      M1000  ; CONV'S  AUTOMODE
      LD=     K1130 D1000  ; CONV'S  STEP SEQ
      OR=     K2130 D1000  ; CONV'S  STEP SEQ
      ANB
      OUT     M1167  ; CONV'1  COMPT
104   LD      M1000  ; CONV'S  AUTOMODE
      LD<=    K1210 D1000  ; CONV'S  STEP SEQ
      AND>=   K1220 D1000  ; CONV'S  STEP SEQ
      LD<=    K2210 D1000  ; CONV'S  STEP SEQ
      AND>=   K2220 D1000  ; CONV'S  STEP SEQ
      ORB
      ANB
      OUT     M1265  ; CONV'2  TRANSFERREQUEST
120   LD      M1000  ; CONV'S  AUTOMODE
      LD=     K1220 D1000  ; CONV'S  STEP SEQ
      OR=     K2220 D1000  ; CONV'S  STEP SEQ
      ANB
      OUT     M1266  ; CONV'2  BUSY
129   LD      M1000  ; CONV'S  AUTOMODE
      LD=     K1230 D1000  ; CONV'S  STEP SEQ
      OR=     K2230 D1000  ; CONV'S  STEP SEQ
      ANB
      OUT     M1267  ; CONV'2  COMPT
138   LD      M1000  ; CONV'S  AUTOMODE
      LD<=    K1310 D1000  ; CONV'S  STEP SEQ
      AND>=   K1320 D1000  ; CONV'S  STEP SEQ
      LD<=    K2310 D1000  ; CONV'S  STEP SEQ
      AND>=   K2320 D1000  ; CONV'S  STEP SEQ
      ORB
      ANB
      OUT     M1365  ; CONV'3  TRANSFERREQUEST
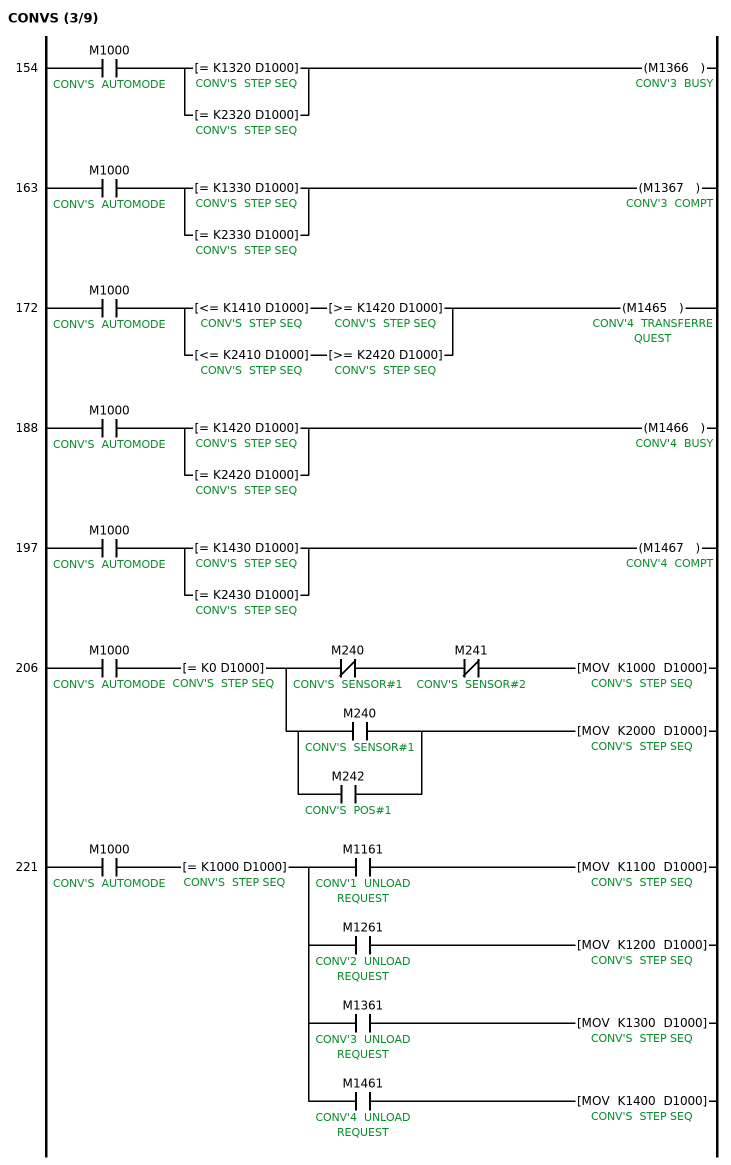
154   LD      M1000  ; CONV'S  AUTOMODE
      LD=     K1320 D1000  ; CONV'S  STEP SEQ
      OR=     K2320 D1000  ; CONV'S  STEP SEQ
      ANB
      OUT     M1366  ; CONV'3  BUSY
163   LD      M1000  ; CONV'S  AUTOMODE
      LD=     K1330 D1000  ; CONV'S  STEP SEQ
      OR=     K2330 D1000  ; CONV'S  STEP SEQ
      ANB
      OUT     M1367  ; CONV'3  COMPT
172   LD      M1000  ; CONV'S  AUTOMODE
      LD<=    K1410 D1000  ; CONV'S  STEP SEQ
      AND>=   K1420 D1000  ; CONV'S  STEP SEQ
      LD<=    K2410 D1000  ; CONV'S  STEP SEQ
      AND>=   K2420 D1000  ; CONV'S  STEP SEQ
      ORB
      ANB
      OUT     M1465  ; CONV'4  TRANSFERREQUEST
188   LD      M1000  ; CONV'S  AUTOMODE
      LD=     K1420 D1000  ; CONV'S  STEP SEQ
      OR=     K2420 D1000  ; CONV'S  STEP SEQ
      ANB
      OUT     M1466  ; CONV'4  BUSY
197   LD      M1000  ; CONV'S  AUTOMODE
      LD=     K1430 D1000  ; CONV'S  STEP SEQ
      OR=     K2430 D1000  ; CONV'S  STEP SEQ
      ANB
      OUT     M1467  ; CONV'4  COMPT
206   LD      M1000  ; CONV'S  AUTOMODE
      AND=    K0 D1000  ; CONV'S  STEP SEQ
      MPS
      ANI     M240  ; CONV'S  SENSOR#1
      ANI     M241  ; CONV'S  SENSOR#2
      MOV     K1000 D1000
      MPP
      LD      M240  ; CONV'S  SENSOR#1
      OR      M242  ; CONV'S  POS#1
      ANB
      MOV     K2000 D1000
221   LD      M1000  ; CONV'S  AUTOMODE
      AND=    K1000 D1000  ; CONV'S  STEP SEQ
      MPS
      AND     M1161  ; CONV'1  UNLOAD  REQUEST
      MOV     K1100 D1000
      MRD
      AND     M1261  ; CONV'2  UNLOAD  REQUEST
      MOV     K1200 D1000
      MRD
      AND     M1361  ; CONV'3  UNLOAD  REQUEST
      MOV     K1300 D1000
      MPP
      AND     M1461  ; CONV'4  UNLOAD  REQUEST
      MOV     K1400 D1000
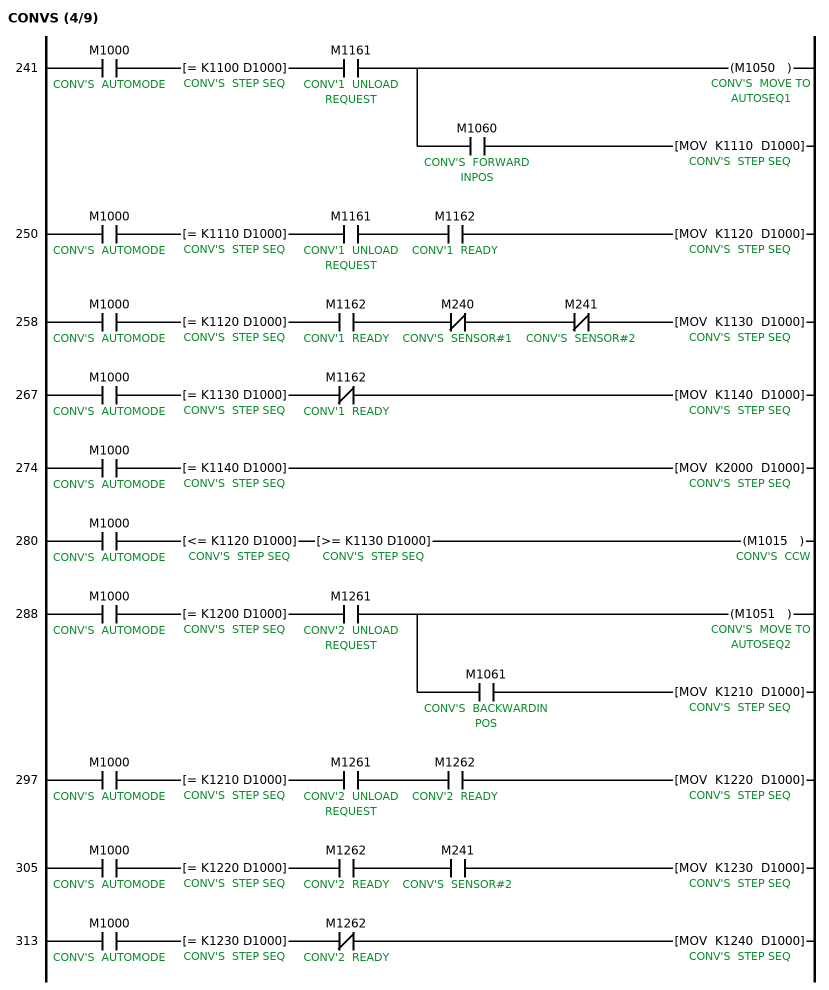
241   LD      M1000  ; CONV'S  AUTOMODE
      AND=    K1100 D1000  ; CONV'S  STEP SEQ
      AND     M1161  ; CONV'1  UNLOAD  REQUEST
      OUT     M1050  ; CONV'S  MOVE TO AUTOSEQ1
      AND     M1060  ; CONV'S  FORWARD INPOS
      MOV     K1110 D1000
250   LD      M1000  ; CONV'S  AUTOMODE
      AND=    K1110 D1000  ; CONV'S  STEP SEQ
      AND     M1161  ; CONV'1  UNLOAD  REQUEST
      AND     M1162  ; CONV'1  READY
      MOV     K1120 D1000
258   LD      M1000  ; CONV'S  AUTOMODE
      AND=    K1120 D1000  ; CONV'S  STEP SEQ
      AND     M1162  ; CONV'1  READY
      ANI     M240  ; CONV'S  SENSOR#1
      ANI     M241  ; CONV'S  SENSOR#2
      MOV     K1130 D1000
267   LD      M1000  ; CONV'S  AUTOMODE
      AND=    K1130 D1000  ; CONV'S  STEP SEQ
      ANI     M1162  ; CONV'1  READY
      MOV     K1140 D1000
274   LD      M1000  ; CONV'S  AUTOMODE
      AND=    K1140 D1000  ; CONV'S  STEP SEQ
      MOV     K2000 D1000
280   LD      M1000  ; CONV'S  AUTOMODE
      AND<=   K1120 D1000  ; CONV'S  STEP SEQ
      AND>=   K1130 D1000  ; CONV'S  STEP SEQ
      OUT     M1015  ; CONV'S  CCW
288   LD      M1000  ; CONV'S  AUTOMODE
      AND=    K1200 D1000  ; CONV'S  STEP SEQ
      AND     M1261  ; CONV'2  UNLOAD  REQUEST
      OUT     M1051  ; CONV'S  MOVE TO AUTOSEQ2
      AND     M1061  ; CONV'S  BACKWARDINPOS
      MOV     K1210 D1000
297   LD      M1000  ; CONV'S  AUTOMODE
      AND=    K1210 D1000  ; CONV'S  STEP SEQ
      AND     M1261  ; CONV'2  UNLOAD  REQUEST
      AND     M1262  ; CONV'2  READY
      MOV     K1220 D1000
305   LD      M1000  ; CONV'S  AUTOMODE
      AND=    K1220 D1000  ; CONV'S  STEP SEQ
      AND     M1262  ; CONV'2  READY
      AND     M241  ; CONV'S  SENSOR#2
      MOV     K1230 D1000
313   LD      M1000  ; CONV'S  AUTOMODE
      AND=    K1230 D1000  ; CONV'S  STEP SEQ
      ANI     M1262  ; CONV'2  READY
      MOV     K1240 D1000
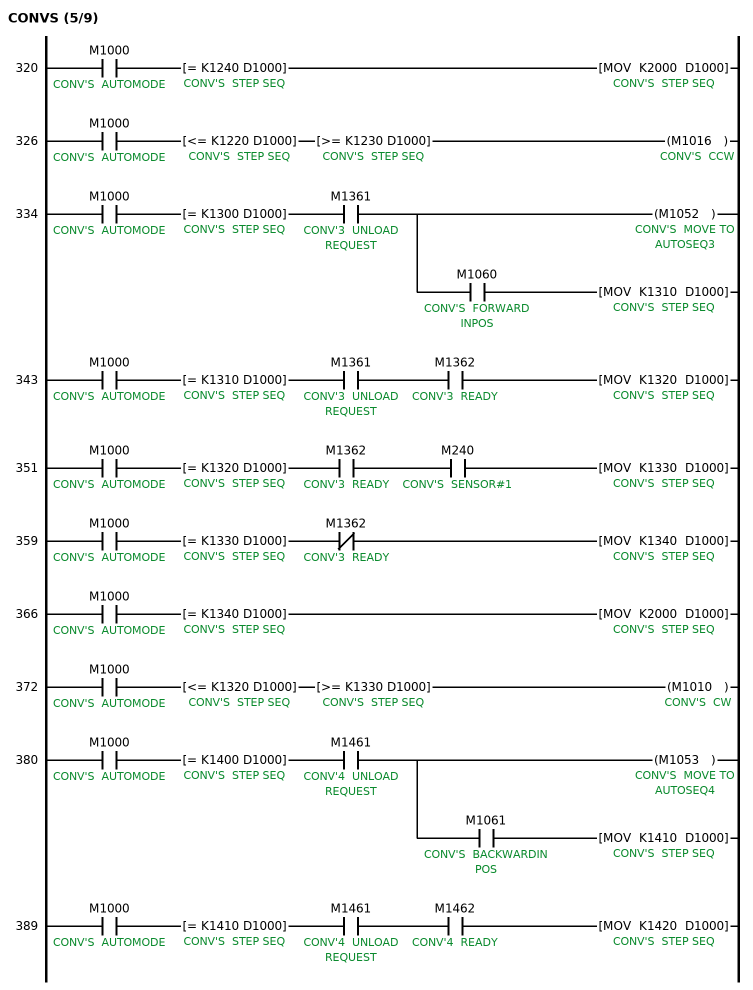
320   LD      M1000  ; CONV'S  AUTOMODE
      AND=    K1240 D1000  ; CONV'S  STEP SEQ
      MOV     K2000 D1000
326   LD      M1000  ; CONV'S  AUTOMODE
      AND<=   K1220 D1000  ; CONV'S  STEP SEQ
      AND>=   K1230 D1000  ; CONV'S  STEP SEQ
      OUT     M1016  ; CONV'S  CCW
334   LD      M1000  ; CONV'S  AUTOMODE
      AND=    K1300 D1000  ; CONV'S  STEP SEQ
      AND     M1361  ; CONV'3  UNLOAD  REQUEST
      OUT     M1052  ; CONV'S  MOVE TO AUTOSEQ3
      AND     M1060  ; CONV'S  FORWARD INPOS
      MOV     K1310 D1000
343   LD      M1000  ; CONV'S  AUTOMODE
      AND=    K1310 D1000  ; CONV'S  STEP SEQ
      AND     M1361  ; CONV'3  UNLOAD  REQUEST
      AND     M1362  ; CONV'3  READY
      MOV     K1320 D1000
351   LD      M1000  ; CONV'S  AUTOMODE
      AND=    K1320 D1000  ; CONV'S  STEP SEQ
      AND     M1362  ; CONV'3  READY
      AND     M240  ; CONV'S  SENSOR#1
      MOV     K1330 D1000
359   LD      M1000  ; CONV'S  AUTOMODE
      AND=    K1330 D1000  ; CONV'S  STEP SEQ
      ANI     M1362  ; CONV'3  READY
      MOV     K1340 D1000
366   LD      M1000  ; CONV'S  AUTOMODE
      AND=    K1340 D1000  ; CONV'S  STEP SEQ
      MOV     K2000 D1000
372   LD      M1000  ; CONV'S  AUTOMODE
      AND<=   K1320 D1000  ; CONV'S  STEP SEQ
      AND>=   K1330 D1000  ; CONV'S  STEP SEQ
      OUT     M1010  ; CONV'S  CW
380   LD      M1000  ; CONV'S  AUTOMODE
      AND=    K1400 D1000  ; CONV'S  STEP SEQ
      AND     M1461  ; CONV'4  UNLOAD  REQUEST
      OUT     M1053  ; CONV'S  MOVE TO AUTOSEQ4
      AND     M1061  ; CONV'S  BACKWARDINPOS
      MOV     K1410 D1000
389   LD      M1000  ; CONV'S  AUTOMODE
      AND=    K1410 D1000  ; CONV'S  STEP SEQ
      AND     M1461  ; CONV'4  UNLOAD  REQUEST
      AND     M1462  ; CONV'4  READY
      MOV     K1420 D1000
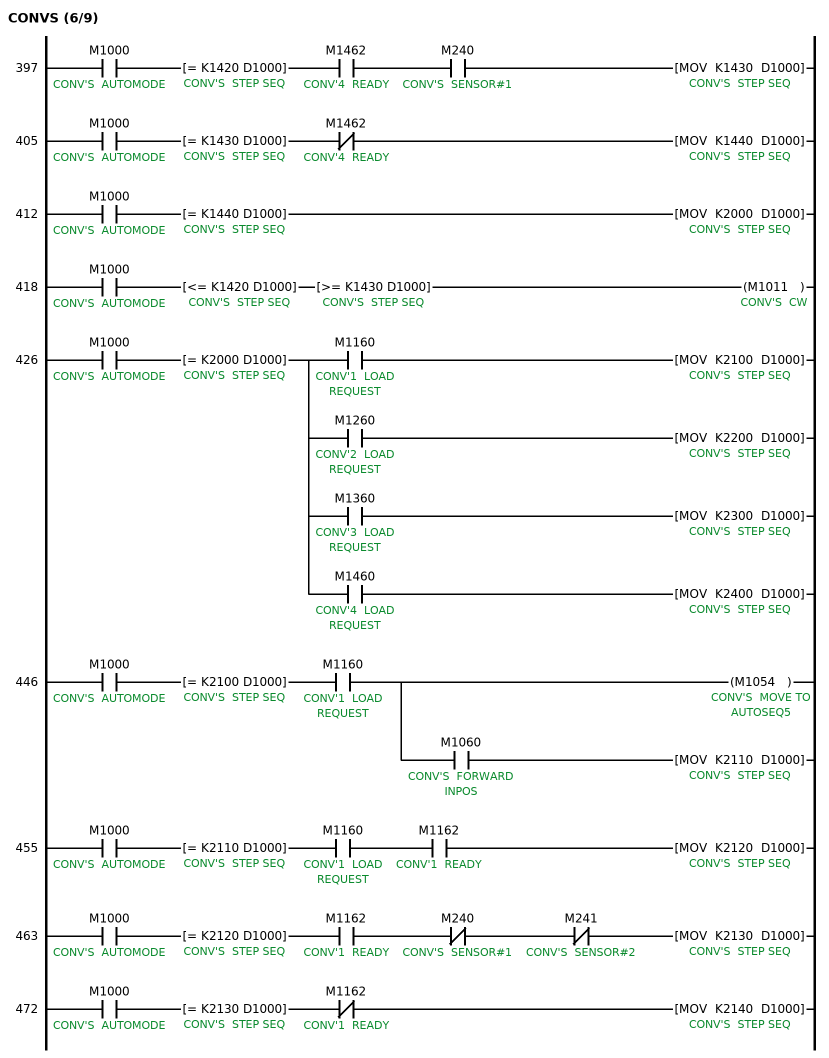
397   LD      M1000  ; CONV'S  AUTOMODE
      AND=    K1420 D1000  ; CONV'S  STEP SEQ
      AND     M1462  ; CONV'4  READY
      AND     M240  ; CONV'S  SENSOR#1
      MOV     K1430 D1000
405   LD      M1000  ; CONV'S  AUTOMODE
      AND=    K1430 D1000  ; CONV'S  STEP SEQ
      ANI     M1462  ; CONV'4  READY
      MOV     K1440 D1000
412   LD      M1000  ; CONV'S  AUTOMODE
      AND=    K1440 D1000  ; CONV'S  STEP SEQ
      MOV     K2000 D1000
418   LD      M1000  ; CONV'S  AUTOMODE
      AND<=   K1420 D1000  ; CONV'S  STEP SEQ
      AND>=   K1430 D1000  ; CONV'S  STEP SEQ
      OUT     M1011  ; CONV'S  CW
426   LD      M1000  ; CONV'S  AUTOMODE
      AND=    K2000 D1000  ; CONV'S  STEP SEQ
      MPS
      AND     M1160  ; CONV'1  LOAD    REQUEST
      MOV     K2100 D1000
      MRD
      AND     M1260  ; CONV'2  LOAD    REQUEST
      MOV     K2200 D1000
      MRD
      AND     M1360  ; CONV'3  LOAD    REQUEST
      MOV     K2300 D1000
      MPP
      AND     M1460  ; CONV'4  LOAD    REQUEST
      MOV     K2400 D1000
446   LD      M1000  ; CONV'S  AUTOMODE
      AND=    K2100 D1000  ; CONV'S  STEP SEQ
      AND     M1160  ; CONV'1  LOAD    REQUEST
      OUT     M1054  ; CONV'S  MOVE TO AUTOSEQ5
      AND     M1060  ; CONV'S  FORWARD INPOS
      MOV     K2110 D1000
455   LD      M1000  ; CONV'S  AUTOMODE
      AND=    K2110 D1000  ; CONV'S  STEP SEQ
      AND     M1160  ; CONV'1  LOAD    REQUEST
      AND     M1162  ; CONV'1  READY
      MOV     K2120 D1000
463   LD      M1000  ; CONV'S  AUTOMODE
      AND=    K2120 D1000  ; CONV'S  STEP SEQ
      AND     M1162  ; CONV'1  READY
      ANI     M240  ; CONV'S  SENSOR#1
      ANI     M241  ; CONV'S  SENSOR#2
      MOV     K2130 D1000
472   LD      M1000  ; CONV'S  AUTOMODE
      AND=    K2130 D1000  ; CONV'S  STEP SEQ
      ANI     M1162  ; CONV'1  READY
      MOV     K2140 D1000
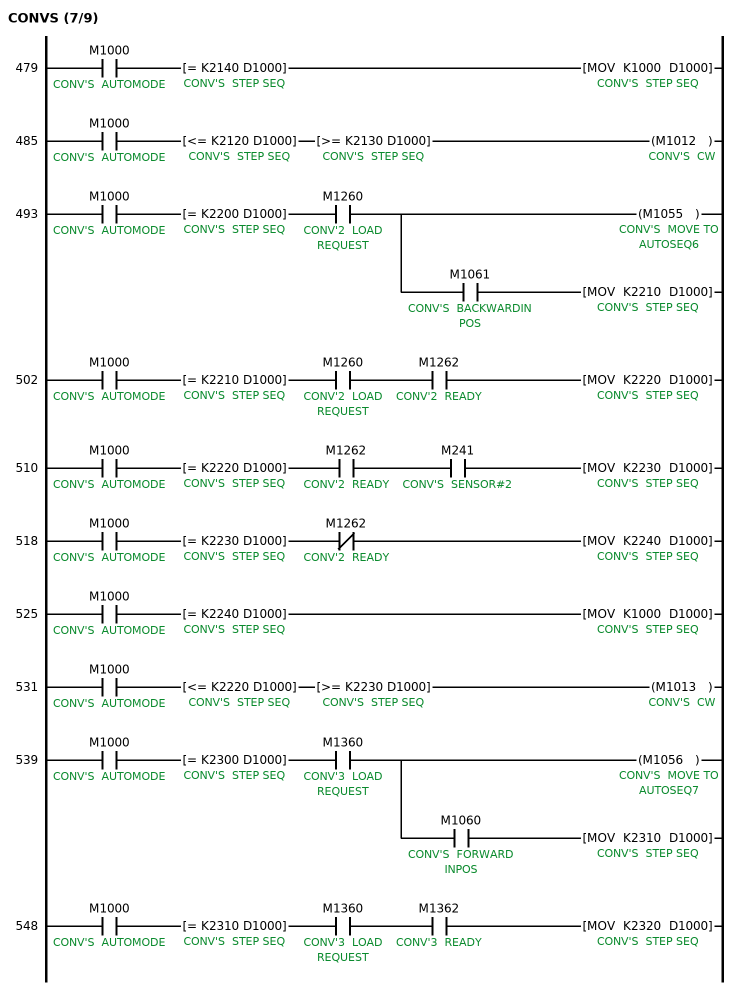
479   LD      M1000  ; CONV'S  AUTOMODE
      AND=    K2140 D1000  ; CONV'S  STEP SEQ
      MOV     K1000 D1000
485   LD      M1000  ; CONV'S  AUTOMODE
      AND<=   K2120 D1000  ; CONV'S  STEP SEQ
      AND>=   K2130 D1000  ; CONV'S  STEP SEQ
      OUT     M1012  ; CONV'S  CW
493   LD      M1000  ; CONV'S  AUTOMODE
      AND=    K2200 D1000  ; CONV'S  STEP SEQ
      AND     M1260  ; CONV'2  LOAD    REQUEST
      OUT     M1055  ; CONV'S  MOVE TO AUTOSEQ6
      AND     M1061  ; CONV'S  BACKWARDINPOS
      MOV     K2210 D1000
502   LD      M1000  ; CONV'S  AUTOMODE
      AND=    K2210 D1000  ; CONV'S  STEP SEQ
      AND     M1260  ; CONV'2  LOAD    REQUEST
      AND     M1262  ; CONV'2  READY
      MOV     K2220 D1000
510   LD      M1000  ; CONV'S  AUTOMODE
      AND=    K2220 D1000  ; CONV'S  STEP SEQ
      AND     M1262  ; CONV'2  READY
      AND     M241  ; CONV'S  SENSOR#2
      MOV     K2230 D1000
518   LD      M1000  ; CONV'S  AUTOMODE
      AND=    K2230 D1000  ; CONV'S  STEP SEQ
      ANI     M1262  ; CONV'2  READY
      MOV     K2240 D1000
525   LD      M1000  ; CONV'S  AUTOMODE
      AND=    K2240 D1000  ; CONV'S  STEP SEQ
      MOV     K1000 D1000
531   LD      M1000  ; CONV'S  AUTOMODE
      AND<=   K2220 D1000  ; CONV'S  STEP SEQ
      AND>=   K2230 D1000  ; CONV'S  STEP SEQ
      OUT     M1013  ; CONV'S  CW
539   LD      M1000  ; CONV'S  AUTOMODE
      AND=    K2300 D1000  ; CONV'S  STEP SEQ
      AND     M1360  ; CONV'3  LOAD    REQUEST
      OUT     M1056  ; CONV'S  MOVE TO AUTOSEQ7
      AND     M1060  ; CONV'S  FORWARD INPOS
      MOV     K2310 D1000
548   LD      M1000  ; CONV'S  AUTOMODE
      AND=    K2310 D1000  ; CONV'S  STEP SEQ
      AND     M1360  ; CONV'3  LOAD    REQUEST
      AND     M1362  ; CONV'3  READY
      MOV     K2320 D1000
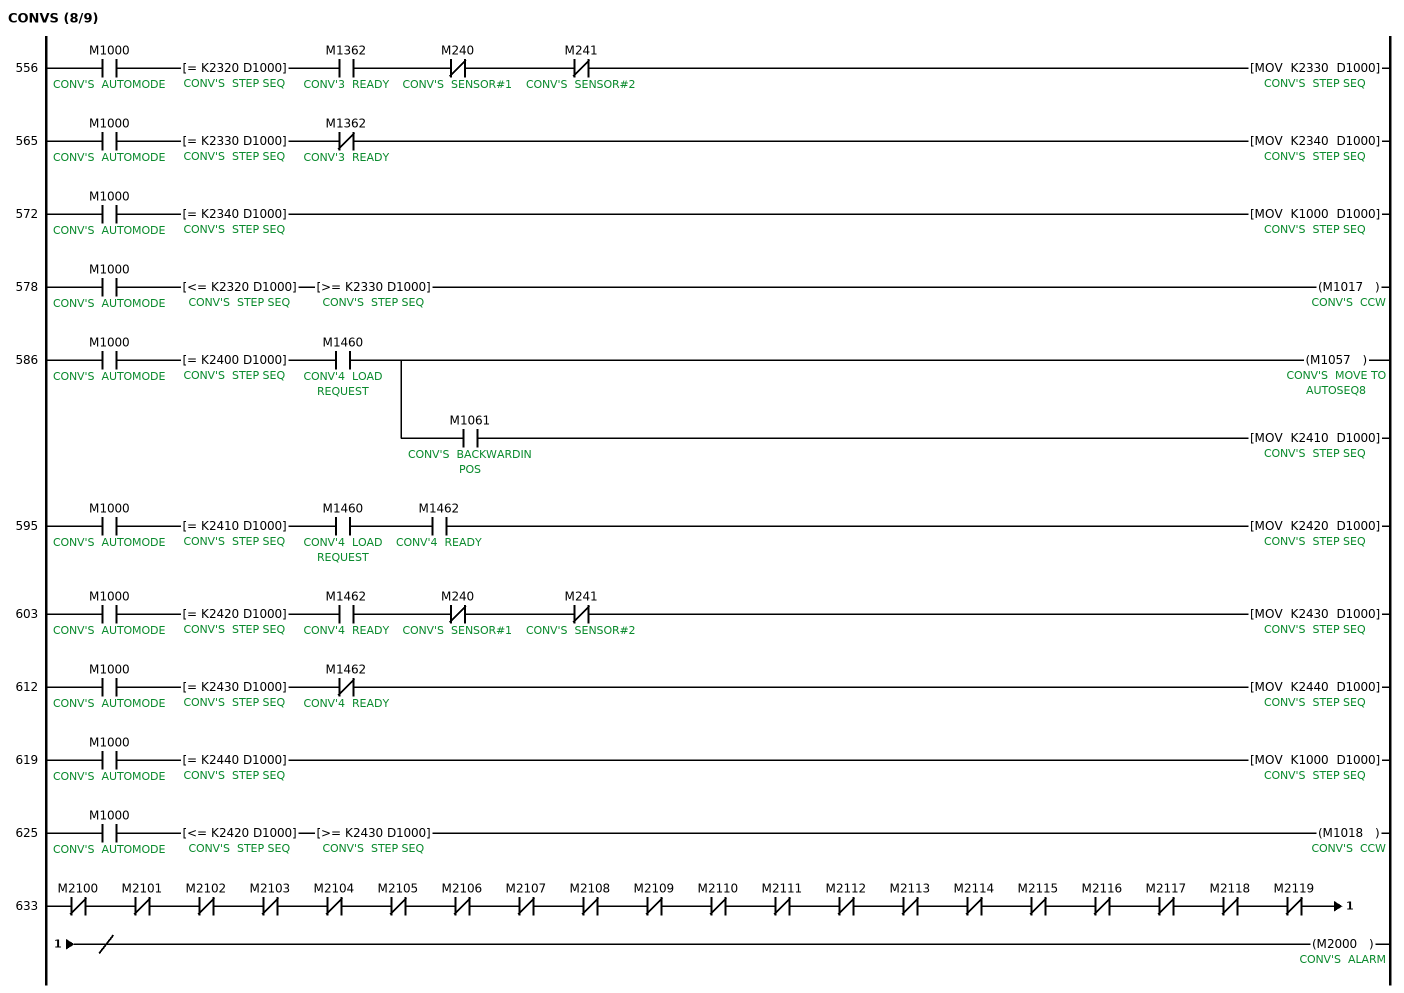
556   LD      M1000  ; CONV'S  AUTOMODE
      AND=    K2320 D1000  ; CONV'S  STEP SEQ
      AND     M1362  ; CONV'3  READY
      ANI     M240  ; CONV'S  SENSOR#1
      ANI     M241  ; CONV'S  SENSOR#2
      MOV     K2330 D1000
565   LD      M1000  ; CONV'S  AUTOMODE
      AND=    K2330 D1000  ; CONV'S  STEP SEQ
      ANI     M1362  ; CONV'3  READY
      MOV     K2340 D1000
572   LD      M1000  ; CONV'S  AUTOMODE
      AND=    K2340 D1000  ; CONV'S  STEP SEQ
      MOV     K1000 D1000
578   LD      M1000  ; CONV'S  AUTOMODE
      AND<=   K2320 D1000  ; CONV'S  STEP SEQ
      AND>=   K2330 D1000  ; CONV'S  STEP SEQ
      OUT     M1017  ; CONV'S  CCW
586   LD      M1000  ; CONV'S  AUTOMODE
      AND=    K2400 D1000  ; CONV'S  STEP SEQ
      AND     M1460  ; CONV'4  LOAD    REQUEST
      OUT     M1057  ; CONV'S  MOVE TO AUTOSEQ8
      AND     M1061  ; CONV'S  BACKWARDINPOS
      MOV     K2410 D1000
595   LD      M1000  ; CONV'S  AUTOMODE
      AND=    K2410 D1000  ; CONV'S  STEP SEQ
      AND     M1460  ; CONV'4  LOAD    REQUEST
      AND     M1462  ; CONV'4  READY
      MOV     K2420 D1000
603   LD      M1000  ; CONV'S  AUTOMODE
      AND=    K2420 D1000  ; CONV'S  STEP SEQ
      AND     M1462  ; CONV'4  READY
      ANI     M240  ; CONV'S  SENSOR#1
      ANI     M241  ; CONV'S  SENSOR#2
      MOV     K2430 D1000
612   LD      M1000  ; CONV'S  AUTOMODE
      AND=    K2430 D1000  ; CONV'S  STEP SEQ
      ANI     M1462  ; CONV'4  READY
      MOV     K2440 D1000
619   LD      M1000  ; CONV'S  AUTOMODE
      AND=    K2440 D1000  ; CONV'S  STEP SEQ
      MOV     K1000 D1000
625   LD      M1000  ; CONV'S  AUTOMODE
      AND<=   K2420 D1000  ; CONV'S  STEP SEQ
      AND>=   K2430 D1000  ; CONV'S  STEP SEQ
      OUT     M1018  ; CONV'S  CCW
633   LDI     M2100
      ANI     M2101
      ANI     M2102
      ANI     M2103
      ANI     M2104
      ANI     M2105
      ANI     M2106
      ANI     M2107
      ANI     M2108
      ANI     M2109
      ANI     M2110
      ANI     M2111
      ANI     M2112
      ANI     M2113
      ANI     M2114
      ANI     M2115
      ANI     M2116
      ANI     M2117
      ANI     M2118
      ANI     M2119
      INV
      OUT     M2000  ; CONV'S  ALARM
